// TIA Portal V20 export
TYPE "typeMTPModuleTypePackageRevision"
TITLE = MTP versioning / MTP-Versionierung
// MTP version information / MTP Versionsinformation
   STRUCT
      ModuleTypePackageRevision { ExternalAccessible := 'False'; ExternalVisible := 'False'; ExternalWritable := 'False'} : String := '0.0.1';   // ModuleTypePackageRevision; Schema: Major.Minor.Patch / ModuleTypePackageRevision; scheme: Major.Minor.Patch
   END_STRUCT;
END_TYPE
